Fanuc KAREL source: ERR_DATA.kl

PROGRAM T
%NOLOCKGROUP
VAR
 v0 : INTEGER
 v1 : INTEGER
 v2 : STRING[40]
 v3 : INTEGER
 v4 : STRING[40]
 v5 : INTEGER
 v6 : INTEGER
 v7 : STRING[40]
BEGIN
 ERR_DATA(v0, v1, v2, v3, v4, v5, v6, v7)
END T
